// TIA Portal V18 export
TYPE "typeSpotList"
// stored: IsFailsafeCompliant false
   STRUCT
      N : Int;
      pos_AR : Array[1..30] of "typePositions";
   END_STRUCT;
END_TYPE
